Staubli VAL3: ioLinks.pgx

program ioLinks()
begin
  dioLink(iEmergencyIn,io:EmergencyIn)
  dioLink(iSchock,io:Schock)
  dioLink(iGripOpen,io:GripOpen)
  dioLink(iGripClosed,io:GripClosed)
  dioLink(iRack1,io:Rack1)
  dioLink(iRack2,io:Rack2)
  dioLink(iRack3,io:Rack3)
  dioLink(iRack4,io:Rack4)
  dioLink(iIdent1,io:Ident1)
  dioLink(iIdent2,io:Ident2)
  dioLink(iIdent3,io:Ident3)
  dioLink(iPressureSensor,io:PressureSensor)
  dioLink(iCryoShortIn,io:CryoShortIn)
  dioLink(iCryoLongIn,io:CryoLongIn)
  dioLink(iPilatusPos,io:PilatusPos)
  dioLink(iPlate1,io:Plate1)
  dioLink(iPlate2,io:Plate2)
  dioLink(iPlate3,io:Plate3)
  dioLink(iLevelFault,io:LevelFault)
  dioLink(iLevel1,io:Level1)
  dioLink(iLevel2,io:Level2)
  dioLink(iLevel3,io:Level3)
  dioLink(iLevel4,io:Level4)
  dioLink(iLevel5,io:Level5)
  dioLink(iLidClosed,io:LidClosed)
  dioLink(iFluorOpen,io:FluorOpen)
  dioLink(iFluorClosed,io:FluorClosed)
  dioLink(iHeaterStatus,io:HeaterStatus)
  dioLink(iSampleStatus,io:SampleStatus)
  dioLink(oResetFault,io:ResetFault)
  dioLink(oEmergencyOut,io:EmergencyOut)
  dioLink(oCryoShortOut,io:CryoShortOut)
  dioLink(oCryoLongOut,io:CryoLongOut)
  dioLink(oFluorDet,io:FluorDet)
  dioLink(oPilatusCover,io:PilatusCover)
  dioLink(oLid,io:Lid)
  dioLink(oHeater,io:Heater)
  dioLink(oShutter,io:Shutter)
  dioLink(oVacuumValve,io:VacuumValve)
  dioLink(oGripCmd,io:valve1)
  dioLink(oGripCmd2,io:valve2)
  dioLink(oSample,io:Sample)
  aioLink(aLight1,io:Light1)
  aioLink(aLight2,io:Light2)
  aioLink(aLight3,io:Light3)
  aioLink(aHeaterTime,io:HeaterTime)
end
